(* CODESYS project SPT_EtherCat.library
   Author: SPT
   Version: 4.0.1
   Title: SPT EtherCat
   Placeholder: SPT EtherCat
   Company: Beckhoff Automation LLC

Project tree, tasks and I/O mapping:
  libraries: SPT Base Types, * (Beckhoff Automation LLC); SPT Event Logger, * (Beckhoff Automation LLC); Tc2_EtherCAT, * (Beckhoff Automation GmbH); Tc2_Standard, * (Beckhoff Automation GmbH); Tc2_System, * (Beckhoff Automation GmbH); Tc3_EventLogger, * (Beckhoff Automation GmbH); Tc3_Module, * (Beckhoff Automation GmbH)
  DUT/
    data type ST_EtherCatMaster_Command
    data type ST_EtherCatMaster_Config
    data type ST_EtherCatMaster_HMI
    data type ST_EtherCatMaster_Status
    data type ST_EtherCatMasterInfo
    data type ST_EtherCatSyncUnitTaskInfo
  Interface/
    interface I_EtherCatMaster: AmsNetIdEcMaster, ConfiguredSlaveCount, ConfiguredSlaveInfo, RegisterSyncUnit
    interface I_SyncUnitTask: IsHotConnect, NumberOfSlaves, SyncUnitName
  Project Information/
    function F_GetCompany [ST]
    function F_GetTitle [ST]
    function F_GetVersion [ST]
  Version/
    global variables Global_Version
  function block FB_Component_EtherCatMaster [ST]: CreateEvents, Monitoring, Reset, CyclicLogic, AmsNetIdEcMaster, ConfiguredSlaveCount, ConfiguredSlaveInfo, RegisterSyncUnit, FramesWcStatesOk, HMICommunication, Initialize, LookupMasterDevState, LookupSlaveDevState, MasterState, SlaveState
  function block FB_SyncUnitTask [ST]: CyclicLogic, IsHotConnect, NumberOfSlaves, SyncUnitName, FB_exit, FB_init, Initialize
  00000000-0000-0000-0000-000000000000|LICENSE
  LICENSE
  global variables Parameter_EtherCatMaster
*)

// DUT/ST_EtherCatMaster_Command
TYPE ST_EtherCatMaster_Command :
	STRUCT
	END_STRUCT
END_TYPE

// DUT/ST_EtherCatMaster_Config
TYPE ST_EtherCatMaster_Config :
	STRUCT
	END_STRUCT
END_TYPE

// DUT/ST_EtherCatMaster_HMI
TYPE ST_EtherCatMaster_HMI :
	STRUCT
		Config	: ST_EtherCatMaster_Config;
		Command : ST_EtherCatMaster_Command;
		Status	: ST_EtherCatMaster_Status;
	END_STRUCT
END_TYPE

// DUT/ST_EtherCatMaster_Status
TYPE ST_EtherCatMaster_Status :
	STRUCT
		AmsNetID			: T_AMSNETID;
		CfgSlaveCount		: UINT;
		EcSlavesState		: ARRAY[0..EC_MAX_SLAVES] OF ST_EcSlaveState;
		ConfiguredSlaveInfo : ARRAY[0..EC_MAX_SLAVES] OF ST_EcSlaveConfigData;
		EcSlaveTopologyInfo : ARRAY[0..EC_MAX_SLAVES] OF ST_TopologyDataEx;
	END_STRUCT
END_TYPE

// DUT/ST_EtherCatMasterInfo
TYPE ST_EtherCatMasterInfo :
	STRUCT
		AmsNetID	  AT %I* : AMSNETID;
		DevID		  AT %I* : UINT;
		DevState	  AT %I* : UINT;
		ChangeCount	  AT %I* : UINT;
		SlaveCount	  AT %I* : UINT;
		CfgSlaveCount AT %I* : UINT;
	END_STRUCT
END_TYPE

// DUT/ST_EtherCatSyncUnitTaskInfo
TYPE ST_EtherCatSyncUnitTaskInfo :
	STRUCT
		WcState	   AT %I* : BIT;
		ObjectId   AT %I* : OTCID;
		State	   AT %I* : UINT;
		SlaveCount AT %I* : UINT;
	END_STRUCT
END_TYPE

// Version/Global_Version
{attribute 'TcGenerated'}
{attribute 'no-analysis'}
{attribute 'linkalways'}
// This function has been automatically generated from the project information.
VAR_GLOBAL CONSTANT
	{attribute 'const_non_replaced'}
	stLibVersion_SPT_EtherCat : ST_LibVersion := (iMajor := 4, iMinor := 0, iBuild := 1, iRevision := 0, nFlags := 0, sVersion := '4.0.1');
END_VAR

// Parameter_EtherCatMaster
{attribute 'qualified_only'}
VAR_GLOBAL CONSTANT
	SYNC_UNIT_TASKS_PER_MASTER : UDINT := 10;	// Max Count of Sync Units per Master
	FRAMES_MAX				   : UDINT := 10;	// Max Count of Frames to Diagnose
	START_UP_TIME			   : TIME  := T#1S; // Time to Startup EtherCat Master Diagnostic at initial startup
END_VAR

// Interface/I_EtherCatMaster
INTERFACE I_EtherCatMaster EXTENDS I_ComponentBase

PROPERTY AmsNetIdEcMaster : T_AMSNETID
GET
END_GET
END_PROPERTY

PROPERTY ConfiguredSlaveCount : UINT
GET
END_GET
END_PROPERTY

PROPERTY ConfiguredSlaveInfo : REFERENCE TO ARRAY[0..EC_MAX_SLAVES] OF ST_EcSlaveConfigData
GET
END_GET
END_PROPERTY

METHOD RegisterSyncUnit : BOOL
VAR_INPUT
	ipSyncUnitTask : I_SyncUnitTask;
END_VAR
END_METHOD

END_INTERFACE

// Interface/I_SyncUnitTask
INTERFACE I_SyncUnitTask EXTENDS I_CyclicFB

PROPERTY IsHotConnect : BOOL
GET
END_GET
SET
END_SET
END_PROPERTY

PROPERTY PUBLIC NumberOfSlaves : UINT
GET
END_GET
END_PROPERTY

PROPERTY SyncUnitName : STRING(63)
GET
END_GET
END_PROPERTY

END_INTERFACE

// Project Information/F_GetCompany
// This function has been automatically generated from the project information.
{attribute 'signature_flag' := '1073741824'}
{attribute 'TcGenerated'}
{attribute 'no-analysis'}
FUNCTION F_GetCompany : WSTRING
VAR_INPUT
	
END_VAR

F_GetCompany := "Beckhoff Automation LLC";

END_FUNCTION

// Project Information/F_GetTitle
// This function has been automatically generated from the project information.
{attribute 'signature_flag' := '1073741824'}
{attribute 'TcGenerated'}
{attribute 'no-analysis'}
FUNCTION F_GetTitle : WSTRING
VAR_INPUT
	
END_VAR

F_GetTitle := "SPT EtherCat";

END_FUNCTION

// Project Information/F_GetVersion
// This function has been automatically generated from the project information.
{attribute 'signature_flag' := '1073741824'}
{attribute 'TcGenerated'}
{attribute 'no-analysis'}
FUNCTION F_GetVersion : ST_LibVersion
VAR_INPUT
	
END_VAR

F_GetVersion.iMajor := 4;
F_GetVersion.iMinor := 0;
F_GetVersion.iBuild := 1;
F_GetVersion.iRevision := 0;
F_GetVersion.sVersion := '4.0.1';
F_GetVersion.nFlags := 0;

END_FUNCTION

// FB_Component_EtherCatMaster
{attribute 'no_explicit_call' := 'do not call this POU directly'}
FUNCTION_BLOCK FB_Component_EtherCatMaster EXTENDS FB_ComponentBase IMPLEMENTS I_EtherCatMaster
VAR
	// Connections
	EtherCatMaster	   : ST_EtherCatMasterInfo;
	FrmXWcState AT %I* : ARRAY[0..(Parameter_EtherCatMaster.FRAMES_MAX - 1)] OF WORD; // link to task related ethercat frame state (Frm2WcState)

	// Internal Variables	
	_AmsNetIdEcMaster	 : T_AMSNETID;
	GetSlaveTopologyInfo : FB_EcGetSlaveTopologyInfo;
	EcGetAllSlaveStates	 : FB_EcGetAllSlaveStates;
	GetMasterFrameCount	 : FB_EcMasterFrameCount;
	LastFramesWcStatesOk : BOOL;
	EcSlavesState		 : ARRAY[0..EC_MAX_SLAVES] OF ST_EcSlaveState;
	EcSlaveTopologyInfo	 : ARRAY[0..EC_MAX_SLAVES] OF ST_TopologyDataEx;
	GetConfiguredSlaves	 : FB_EcGetConfSlaves;
	_ConfiguredSlaveInfo : ARRAY[0..EC_MAX_SLAVES] OF ST_EcSlaveConfigData;
	i					 : UDINT;

	// HMI
	EtherCatMaster_HMI : ST_EtherCatMaster_HMI;

	// Sync Units per Master
	SyncUnitTask : ARRAY[1..Parameter_EtherCatMaster.SYNC_UNIT_TASKS_PER_MASTER] OF I_SyncUnitTask;

	(*Sequence*)
	SlaveSeq			 : UINT;
	RunSlaveDiag		 : BOOL;
	LastChangeCount		 : UINT := 0;
	LastSlaveCount		 : UINT := 0;
	LastMasterState		 : UINT := 0;
	ErrorMaster			 : BOOL;
	WarningSlaveDisabled : BOOL;
	ErrorSlave			 : BOOL;
	FaultedSlave		 : UINT;

	// Alarms
	ComponentEtherCatDiagAlarms : ARRAY[1..COMPONENT_ETHERCAT_DIAG_ALARM_COUNT] OF FB_TcAlarm;
END_VAR

VAR CONSTANT
	COMPONENT_ETHERCAT_DIAG_ALARM_COUNT : UDINT := 20;
END_VAR

METHOD PROTECTED CreateEvents

// This method is called by Initialize() as required
F_CreateAllEventsInClass(Alarms		:= ComponentEtherCatDiagAlarms,
						 ClassSize	:= SIZEOF(TC_EVENTS.EtherCatDiagnostics),
						 pInitEvent := ADR(TC_EVENTS.EtherCatDiagnostics.InitReferenceEvent),
						 Prefix		:= Name);

SUPER^.CreateEvents();
END_METHOD

// Provides basic error detection and event handling for this component
METHOD PROTECTED Monitoring

// This method is called cyclically by CyclicLogic()
SUPER^.Monitoring();

(*EtherCat Messages*)
IF ErrorSlave AND (_ErrorId = 999) AND NOT ComponentEtherCatDiagAlarms[E_EtherCatDiagnostics.ReadSlave].bRaised THEN
	RaiseEventWithStrings(ComponentEtherCatDiagAlarms[E_EtherCatDiagnostics.ReadSlave], '', '');
ELSIF NOT ErrorSlave AND ComponentEtherCatDiagAlarms[E_EtherCatDiagnostics.ReadSlave].bRaised THEN
	ComponentEtherCatDiagAlarms[E_EtherCatDiagnostics.ReadSlave].Clear(0, 0);
END_IF

IF ErrorMaster AND NOT ComponentEtherCatDiagAlarms[E_EtherCatDiagnostics.MasterError].bRaised THEN
	RaiseAlarmWithStrings(ComponentEtherCatDiagAlarms[E_EtherCatDiagnostics.MasterError], LookupMasterDevState(EtherCatMaster.DevState), '');
END_IF

IF ErrorSlave AND NOT ComponentEtherCatDiagAlarms[E_EtherCatDiagnostics.SlaveError].bRaised THEN
	RaiseAlarmWithStrings(ComponentEtherCatDiagAlarms[E_EtherCatDiagnostics.SlaveError], _ConfiguredSlaveInfo[FaultedSlave].sName, LookupSlaveDevState(FaultedSlave));
END_IF

IF WarningSlaveDisabled AND NOT ComponentEtherCatDiagAlarms[E_EtherCatDiagnostics.SlaveDisabled].bRaised THEN
	RaiseEventWithStrings(ComponentEtherCatDiagAlarms[E_EtherCatDiagnostics.SlaveDisabled], '', '');
ELSIF NOT WarningSlaveDisabled AND ComponentEtherCatDiagAlarms[E_EtherCatDiagnostics.SlaveDisabled].bRaised THEN
	ComponentEtherCatDiagAlarms[E_EtherCatDiagnostics.SlaveDisabled].Clear(0, 0);
END_IF

_CurrentAlarmSeverity := F_GetMaxSeverityRaised(Alarms := ComponentEtherCatDiagAlarms, CurrentSeverity := _CurrentAlarmSeverity);
END_METHOD

// Clears error flags and error IDs for this component
METHOD PUBLIC Reset : BOOL
F_ClearAllEventsInClass(ComponentEtherCatDiagAlarms);
Reset				 := SUPER^.Reset();
WarningSlaveDisabled := FALSE;
LastMasterState		 := 0;
LastChangeCount		 := 0;
LastSlaveCount		 := 0;
_Error				 := FALSE;
_ErrorId			 := 0;
SlaveSeq			 := 0;
RunSlaveDiag		 := FALSE;
END_METHOD

// This method serves as the entry point for all underlying FB logic
METHOD PUBLIC CyclicLogic

// This method should be called cyclically by descendant function blocks by invoking SUPER^.CyclicLogic().  Alternatively, the contents of this method could be reimplemented entirely in which case a call to this method would not be necessary.
IF NOT _InitComplete THEN
	_InitComplete := Initialize();
	RETURN;
END_IF

(* Main Component Signals *)
IF _Simulate THEN
	_Busy	 := FALSE;
	_Error	 := FALSE;
	_ErrorId := 0;
ELSE
	// Initiate Detection of Change
	IF NOT _Busy THEN
		IF (LastChangeCount <> EtherCatMaster.ChangeCount) THEN // Master Change count changed
			RunSlaveDiag := TRUE;
		ELSIF ((EtherCatMaster.CfgSlaveCount <> EtherCatMaster.SlaveCount) AND (LastSlaveCount <> EtherCatMaster.SlaveCount)) THEN // Slave Count changed
			RunSlaveDiag := TRUE;
		ELSIF FramesWcStatesOk() <> LastFramesWcStatesOk THEN // Frame WC state changed
			RunSlaveDiag := TRUE;
		END_IF

		IF RunSlaveDiag THEN // Update Change
			LastChangeCount		 := EtherCatMaster.ChangeCount;
			LastSlaveCount		 := EtherCatMaster.SlaveCount;
			LastFramesWcStatesOk := FramesWcStatesOk();
		END_IF
	END_IF

	// Get slave topology info
	GetSlaveTopologyInfo(sNetId	  := _AmsNetIdEcMaster,
						 pAddrBuf := ADR(EcSlaveTopologyInfo),
						 cbBufLen := SIZEOF(EcSlaveTopologyInfo),
						 tTimeout := T#5S);

	// Get all slave states
	EcGetAllSlaveStates(sNetId	  := _AmsNetIdEcMaster,
						pStateBuf := ADR(EcSlavesState),
						cbBufLen  := SIZEOF(EcSlavesState),
						tTimeout  := T#5S);

	// Master State
	MasterState();

	// Slave State
	SlaveState();

	// SyncUnits
	FOR i := 1 TO Parameter_EtherCatMaster.SYNC_UNIT_TASKS_PER_MASTER DO
		IF SyncUnitTask[i] <> 0 THEN
			SyncUnitTask[i].CyclicLogic();
		END_IF
	END_FOR

	// Super
	_Busy  := SlaveSeq <> 0; // Sequence running
	_Error := _Error OR ErrorMaster OR ErrorSlave;
	SUPER^.CyclicLogic();
END_IF
END_METHOD

PROPERTY AmsNetIdEcMaster : T_AMSNETID
GET
AmsNetIdEcMaster := _AmsNetIdEcMaster;
END_GET
END_PROPERTY

PROPERTY ConfiguredSlaveCount : UINT
GET
ConfiguredSlaveCount := EtherCatMaster.CfgSlaveCount;
END_GET
END_PROPERTY

PROPERTY ConfiguredSlaveInfo : REFERENCE TO ARRAY[0..EC_MAX_SLAVES] OF ST_EcSlaveConfigData
GET
ConfiguredSlaveInfo REF= _ConfiguredSlaveInfo;
END_GET
END_PROPERTY

METHOD RegisterSyncUnit : BOOL
VAR_INPUT
	ipSyncUnitTask : I_SyncUnitTask;
END_VAR
FOR i := 1 TO Parameter_EtherCatMaster.SYNC_UNIT_TASKS_PER_MASTER DO
	IF SyncUnitTask[i] = 0 AND ipSyncUnitTask <> 0 THEN
		SyncUnitTask[i]	 := ipSyncUnitTask;
		RegisterSyncUnit := TRUE;
		RETURN;
	END_IF
END_FOR
END_METHOD

METHOD PROTECTED FramesWcStatesOk : BOOL
VAR_INPUT
END_VAR
FramesWcStatesOk := TRUE;
FOR i := 0 TO (GetMasterFrameCount.nFrames - 1) DO
	IF FrmXWcState[i] <> 0 THEN
		FramesWcStatesOk := FALSE;
		EXIT;
	END_IF
END_FOR
END_METHOD

// Provides interlocks for HMI control and updates HMI status information for this component
METHOD PROTECTED HMICommunication

// This method is called cyclically by CyclicLogic()
SUPER^.HMICommunication();

// Status
EtherCatMaster_HMI.Status.CfgSlaveCount		  := EtherCatMaster.CfgSlaveCount;
EtherCatMaster_HMI.Status.AmsNetID			  := _AmsNetIdEcMaster;
EtherCatMaster_HMI.Status.EcSlavesState		  := EcSlavesState;
EtherCatMaster_HMI.Status.ConfiguredSlaveInfo := ConfiguredSlaveInfo;
EtherCatMaster_HMI.Status.EcSlaveTopologyInfo := EcSlaveTopologyInfo;
END_METHOD

// Basic component initialization logic
METHOD PROTECTED Initialize : BOOL;
VAR_INST
	InitializeSequence : UINT := 0;
	Size			   : UDINT;
	StartupTime		   : TON;
END_VAR

// This method is called by CyclicLogic() as required
IF NOT _Error AND NOT (F_GetMappingStatus(ADR(EtherCatMaster.AmsNetID), SIZEOF(EtherCatMaster.AmsNetID)) <> EplcMappingStatus.MS_Unmapped) AND NOT _Simulate THEN
	_Error := TRUE;
	TRACE('Init Failed - AmsNetID mapped to Master!');
END_IF

IF NOT _Error AND NOT (F_GetMappingStatus(ADR(EtherCatMaster.DevID), SIZEOF(EtherCatMaster.DevID)) <> EplcMappingStatus.MS_Unmapped) AND NOT _Simulate THEN
	_Error := TRUE;
	TRACE('Init Failed - DevID mapped to Master!');
END_IF

IF NOT _Error AND NOT (F_GetMappingStatus(ADR(EtherCatMaster.DevState), SIZEOF(EtherCatMaster.DevState)) <> EplcMappingStatus.MS_Unmapped) AND NOT _Simulate THEN
	_Error := TRUE;
	TRACE('Init Failed - DevState mapped to Master!');
END_IF

IF NOT _Error AND NOT (F_GetMappingStatus(ADR(EtherCatMaster.ChangeCount), SIZEOF(EtherCatMaster.ChangeCount)) <> EplcMappingStatus.MS_Unmapped) AND NOT _Simulate THEN
	_Error := TRUE;
	TRACE('Init Failed - ChangeCount mapped to Master!');
END_IF

IF NOT _Error AND NOT (F_GetMappingStatus(ADR(EtherCatMaster.SlaveCount), SIZEOF(EtherCatMaster.SlaveCount)) <> EplcMappingStatus.MS_Unmapped) AND NOT _Simulate THEN
	_Error := TRUE;
	TRACE('Init Failed - CfgSlaveCount mapped to Master!');
END_IF

IF NOT _Error AND NOT (F_GetMappingStatus(ADR(EtherCatMaster.CfgSlaveCount), SIZEOF(EtherCatMaster.CfgSlaveCount)) <> EplcMappingStatus.MS_Unmapped) AND NOT _Simulate THEN
	_Error := TRUE;
	TRACE('Init Failed - CfgSlaveCount mapped to Master!');
END_IF

IF _Error THEN
	RETURN;
END_IF

IF _Simulate THEN
	Initialize := SUPER^.Initialize();
	RETURN;
END_IF

// Get all Slaves
_AmsNetIdEcMaster := F_CreateAmsNetId(EtherCatMaster.AmsNetID);
GetConfiguredSlaves(sNetId				:= _AmsNetIdEcMaster,
					pArrEcConfSlaveInfo := ADR(_ConfiguredSlaveInfo),
					cbBufLen			:= SIZEOF(_ConfiguredSlaveInfo),
					tTimeout			:= T#1S);

// Get Master Frames
GetMasterFrameCount(sNetId := _AmsNetIdEcMaster, tTimeout := T#1S);

// Init Sequence
CASE InitializeSequence OF
	(* Read Slave Info Data *)
	0:
		GetConfiguredSlaves.bExecute := TRUE;
		IF GetConfiguredSlaves.bBusy THEN
			InitializeSequence := InitializeSequence + 10;
		END_IF

	10:
		IF NOT GetConfiguredSlaves.bBusy AND NOT GetConfiguredSlaves.bError THEN
			InitializeSequence := InitializeSequence + 10;
		END_IF

		IF GetConfiguredSlaves.bError THEN
			_Error := TRUE;
			TRACE('Init Failed - Configured EtherCat Slaves could not be read - check linking of EtherCat Master FB!');
			InitializeSequence := 999;
		END_IF

	20: // Get Master Frame Count
		GetMasterFrameCount.bExecute := TRUE;
		IF GetMasterFrameCount.bBusy THEN
			InitializeSequence := InitializeSequence + 10;
		END_IF

	30:
		IF NOT GetMasterFrameCount.bBusy AND NOT GetMasterFrameCount.bError THEN
			// Check Frame Count
			IF GetMasterFrameCount.nFrames > Parameter_EtherCatMaster.FRAMES_MAX THEN
				_Error := TRUE;
				TRACE('Increase of Frame diagnostic array (Parameter_EtherCatMaster.FRAMES_MAX) and link to FrmXWcState!');
				RETURN;
			END_IF

			// Check Frame Linking
			FOR i := 0 TO (GetMasterFrameCount.nFrames - 1) DO
				IF NOT (F_GetMappingStatus(ADR(FrmXWcState[i]), SIZEOF(FrmXWcState[i])) <> EplcMappingStatus.MS_Unmapped) THEN
					_Error := TRUE;
					TRACE('Init Failed - FrmXWcState[x] not mapped to Master!');
					RETURN;
				END_IF
			END_FOR

			// 
			InitializeSequence := InitializeSequence + 10;
		END_IF

		IF GetMasterFrameCount.bError THEN
			_Error := TRUE;
			TRACE('Init Failed - Configured EtherCat Frames could not be read!');
			InitializeSequence := 999;
		END_IF

	40: // Startup time for Ethercat Master	
		StartupTime(IN := TRUE, PT := Parameter_EtherCatMaster.START_UP_TIME);
		IF StartupTime.Q THEN
			InitializeSequence := InitializeSequence + 10;
		END_IF

	50:
		Initialize := SUPER^.Initialize();
END_CASE
END_METHOD

METHOD PROTECTED LookupMasterDevState : STRING
VAR_INPUT
	State : UINT;
END_VAR
IF State.0 THEN
	LookupMasterDevState := 'Link error';
ELSIF State.1 THEN
	LookupMasterDevState := 'I/O locked after link error (I/O reset required)';
ELSIF State.2 THEN
	LookupMasterDevState := 'Link error (redundancy adapter)';
ELSIF State.3 THEN
	LookupMasterDevState := 'Missing one frame (redundancy mode)';
ELSIF State.4 THEN
	LookupMasterDevState := 'Out of send resources (I/O reset required)';
ELSIF State.5 THEN
	LookupMasterDevState := 'Watchdog triggered';
ELSIF State.6 THEN
	LookupMasterDevState := 'Ethernet driver (miniport) NOT found';
ELSIF State.7 THEN
	LookupMasterDevState := 'I/O reset active';
ELSIF State.8 THEN
	LookupMasterDevState := 'At least one device in INIT state';
ELSIF State.9 THEN
	LookupMasterDevState := 'At least one device in PRE-OP state';
ELSIF State.10 THEN
	LookupMasterDevState := 'At least one device in SAFE-OP state';
ELSIF State.11 THEN
	LookupMasterDevState := 'At least one device indicates an error state';
ELSIF State.12 THEN
	LookupMasterDevState := 'DC not in sync';
ELSE
	LookupMasterDevState := 'State not found';
END_IF
END_METHOD

METHOD PROTECTED LookupSlaveDevState : STRING
VAR_INPUT
	Slave : UINT;
END_VAR

VAR_INST
	DiagByte	: BYTE;
	BitMaskDiag : BYTE := 16#0F;
END_VAR
//_____________________________________________________________________________________________________

(* State *)
BitMaskDiag := 16#0F;
DiagByte	:= EcSlavesState[Slave].deviceState AND BitMaskDiag;
CASE DiagByte OF
	EC_DEVICE_STATE_INIT:
		LookupSlaveDevState := 'Init';

	EC_DEVICE_STATE_PREOP:
		LookupSlaveDevState := 'Pre-op';

	EC_DEVICE_STATE_BOOTSTRAP:
		LookupSlaveDevState := 'Boot';

	EC_DEVICE_STATE_SAFEOP:
		LookupSlaveDevState := 'Safe-op';

	EC_DEVICE_STATE_OP:
		LookupSlaveDevState := 'OP';

ELSE
	LookupSlaveDevState := '';
END_CASE

(* Additional State Bits *)
IF EcSlavesState[Slave].deviceState.4 THEN // EC_DEVICE_STATE_ERROR
	LookupSlaveDevState := CONCAT(LookupSlaveDevState, ' - ');
	LookupSlaveDevState := CONCAT(LookupSlaveDevState, 'State machine error in the EtherCAT slave');
END_IF

IF EcSlavesState[Slave].deviceState.5 THEN // EC_DEVICE_STATE_INVALID_VPRS
	LookupSlaveDevState := CONCAT(LookupSlaveDevState, ' - ');
	LookupSlaveDevState := CONCAT(LookupSlaveDevState, 'Invalid vendor ID');
END_IF

IF EcSlavesState[Slave].deviceState.6 THEN // EC_DEVICE_STATE_INITCMD_ERROR
	LookupSlaveDevState := CONCAT(LookupSlaveDevState, ' - ');
	LookupSlaveDevState := CONCAT(LookupSlaveDevState, 'Error during sending of initialization commands');
END_IF

IF EcSlavesState[Slave].deviceState.7 THEN // EC_DEVICE_STATE_DISABLED
	LookupSlaveDevState := CONCAT(LookupSlaveDevState, ' - ');
	LookupSlaveDevState := CONCAT(LookupSlaveDevState, 'Slave is disabled');
END_IF

//_____________________________________________________________________________________________________

(* Link States *)
IF EcSlavesState[Slave].linkState.0 THEN // EC_LINK_STATE_NOT_PRESENT
	LookupSlaveDevState := CONCAT(LookupSlaveDevState, ' - ');
	LookupSlaveDevState := CONCAT(LookupSlaveDevState, 'No EtherCAT communication with the EtherCAT slave');
END_IF

IF EcSlavesState[Slave].linkState.1 THEN // EC_LINK_STATE_LINK_WITHOUT_COMM
	LookupSlaveDevState := CONCAT(LookupSlaveDevState, ' - ');
	LookupSlaveDevState := CONCAT(LookupSlaveDevState, 'Error AT port X');
END_IF

IF EcSlavesState[Slave].linkState.2 THEN // EC_LINK_STATE_MISSING_LINK
	LookupSlaveDevState := CONCAT(LookupSlaveDevState, ' - ');
	LookupSlaveDevState := CONCAT(LookupSlaveDevState, 'Missing link AT port X');
END_IF

IF EcSlavesState[Slave].linkState.3 THEN // EC_LINK_STATE_ADDITIONAL_LINK
	LookupSlaveDevState := CONCAT(LookupSlaveDevState, ' - ');
	LookupSlaveDevState := CONCAT(LookupSlaveDevState, 'Additional link AT port X');
END_IF

(* Additional State Bits *)
IF EcSlavesState[Slave].linkState.4 THEN // EC_LINK_STATE_PORT_A
	LookupSlaveDevState := CONCAT(LookupSlaveDevState, ' - ');
	LookupSlaveDevState := CONCAT(LookupSlaveDevState, 'Port 0');
END_IF

IF EcSlavesState[Slave].linkState.5 THEN // EC_LINK_STATE_PORT_B
	LookupSlaveDevState := CONCAT(LookupSlaveDevState, ' - ');
	LookupSlaveDevState := CONCAT(LookupSlaveDevState, 'Port 1');
END_IF

IF EcSlavesState[Slave].linkState.6 THEN // EC_LINK_STATE_PORT_C
	LookupSlaveDevState := CONCAT(LookupSlaveDevState, ' - ');
	LookupSlaveDevState := CONCAT(LookupSlaveDevState, 'Port 2');
END_IF

IF EcSlavesState[Slave].linkState.7 THEN // EC_LINK_STATE_PORT_D
	LookupSlaveDevState := CONCAT(LookupSlaveDevState, ' - ');
	LookupSlaveDevState := CONCAT(LookupSlaveDevState, 'Port 3');
END_IF
END_METHOD

METHOD PROTECTED MasterState : BOOL
VAR_INPUT
END_VAR
IF (LastMasterState <> EtherCatMaster.DevState) AND (EtherCatMaster.DevState <> 0) AND (EtherCatMaster.SlaveCount < EtherCatMaster.CfgSlaveCount) THEN
	IF EtherCatMaster.DevState <> 0 THEN // Error in Master
		ErrorMaster := TRUE;
		_ErrorId	:= EtherCatMaster.DevState;
	END_IF
ELSE
	ErrorMaster := FALSE;
END_IF
END_METHOD

METHOD PROTECTED SlaveState : BOOL
VAR_INST
	DiagByte	: BYTE;
	BitMaskDiag : BYTE := 16#0F;
END_VAR
CASE SlaveSeq OF
	(* Wait for start *)
	0:
		EcGetAllSlaveStates.bExecute  := FALSE;
		GetConfiguredSlaves.bExecute  := FALSE;
		GetSlaveTopologyInfo.bExecute := FALSE;
		IF RunSlaveDiag THEN
			RunSlaveDiag		 := FALSE;
			ErrorSlave			 := FALSE; // Reset for re-check
			WarningSlaveDisabled := FALSE;
			SlaveSeq			 := SlaveSeq + 10;
		END_IF

	(* Update Topology*)
	10:
		GetSlaveTopologyInfo.bExecute := TRUE;
		IF GetSlaveTopologyInfo.bBusy THEN
			SlaveSeq := SlaveSeq + 10;
		END_IF

	20:
		IF NOT GetSlaveTopologyInfo.bBusy AND NOT GetSlaveTopologyInfo.bError THEN
			SlaveSeq := SlaveSeq + 10;
		END_IF

		IF GetSlaveTopologyInfo.bError THEN
			SlaveSeq := 999;
		END_IF

	(* Read Slave States *)
	30:
		EcGetAllSlaveStates.bExecute := TRUE;
		IF EcGetAllSlaveStates.bBusy THEN
			SlaveSeq := SlaveSeq + 10;
		END_IF

	40:
		IF NOT EcGetAllSlaveStates.bBusy AND NOT EcGetAllSlaveStates.bError THEN
			SlaveSeq := SlaveSeq + 10;
		END_IF

		IF EcGetAllSlaveStates.bError THEN
			SlaveSeq := 999;
		END_IF

	(* Evaluate Slave Error *)
	50:
		FOR FaultedSlave := 0 TO (EtherCatMaster.CfgSlaveCount - 1) DO
			BitMaskDiag := 16#0F;
			DiagByte	:= EcSlavesState[FaultedSlave].deviceState AND BitMaskDiag;
			IF DiagByte <> EC_DEVICE_STATE_OP AND EcSlaveTopologyInfo[FaultedSlave].nStatusBits.4 = FALSE THEN // No error if hotconnect
				IF EcSlavesState[FaultedSlave].deviceState.7 THEN											   // Slave is Disabled - warning only
					WarningSlaveDisabled := TRUE;
				ELSE
					ErrorSlave := TRUE;
					EXIT;
				END_IF
			END_IF

			BitMaskDiag := 16#0F;
			DiagByte	:= EcSlavesState[FaultedSlave].linkState AND BitMaskDiag;
			IF DiagByte <> EC_LINK_STATE_OK AND EcSlaveTopologyInfo[FaultedSlave].nStatusBits.4 = FALSE THEN // Next slave is in hotconnect group, no error
				ErrorSlave := TRUE;
				EXIT;
			END_IF
		END_FOR

		SlaveSeq := SlaveSeq + 10;

	60:
		SlaveSeq := 0;

	(* Sequence Error*)
	999:
		ErrorSlave := TRUE;
		_ErrorId   := 999;
		SlaveSeq   := 0;
END_CASE
END_METHOD

END_FUNCTION_BLOCK

// FB_SyncUnitTask
{attribute 'no_explicit_call' := 'do not call this POU directly'}
FUNCTION_BLOCK FINAL FB_SyncUnitTask EXTENDS FB_CyclicFB IMPLEMENTS I_SyncUnitTask
VAR
	// IO to Sync Unit Task configuration
	SyncUnitTaskInfo : ST_EtherCatSyncUnitTaskInfo;

	// Internal Variables
	EcGetAllSyncUnitSlaveAddr : FB_EcGetAllSyncUnitSlaveAddr;
	SyncUnitSlaveAddresses	  : POINTER TO UINT;
	SyncUnitSlaveNames		  : POINTER TO STRING(31);
	SyncUnitState			  : (SYNC_UNIT_OK,
		READ_SLAVES,
		POPULATE_SLAVE_NAMES,
		WORKING_COUNTER_ERROR,
		READ_ERROR) := SYNC_UNIT_OK;
	i : UDINT; // Iterator
	j : UDINT; // Iterator

	// Properties
	_SyncUnitName	: STRING(63);
	_NumberOfSlaves : UINT;
	_IsHotConnect	: BOOL;

	// Connection to EtherCat Master
	ipEtherCatMaster : I_EtherCatMaster;

	// Alarm
	SyncUnitAlarm : ARRAY[1..SYNC_UNIT_ALARM_MAX] OF FB_TcAlarm;
END_VAR

VAR
	// Build slave in sync unit collection to display, string limit to 80
	TempSlaveMessage  : STRING;
	SlaveMessagePartA : STRING;
	SlaveMessagePartB : STRING;
END_VAR

VAR CONSTANT
	ERROR_READ_SLAVE_NAMES	   : UDINT := 1;
	ERROR_REGISTER_SYNC_UNIT   : UDINT := 2;
	ERROR_VALID_DATA_SYNC_UNIT : UDINT := 3;
	STRING_LEN				   : INT   := 80;
	SYNC_UNIT_ALARM_MAX		   : UINT  := 3;
END_VAR

METHOD PUBLIC CyclicLogic
VAR_INPUT
END_VAR

VAR_INST
	tempSlaveInfo : REFERENCE TO ARRAY[0..EC_MAX_SLAVES] OF ST_EcSlaveConfigData;
END_VAR
IF NOT _InitComplete THEN
	_InitComplete := Initialize();
	RETURN;
END_IF

// Read SyncUnit Slave Names
tempSlaveInfo REF= ipEtherCatMaster.ConfiguredSlaveInfo;
EcGetAllSyncUnitSlaveAddr(sNetId	:= '',
						  nObjectId := SyncUnitTaskInfo.ObjectId,
						  pAddrBuf	:= SyncUnitSlaveAddresses,
						  cbBufLen	:= (SIZEOF(UINT) * SyncUnitTaskInfo.SlaveCount),
						  tTimeout	:= T#5S,
						  nSlaves	=> _NumberOfSlaves);

EcGetAllSyncUnitSlaveAddr.bExecute := FALSE;

// Sync Unit States
CASE SyncUnitState OF
	SYNC_UNIT_OK: // Working counter error detected on this sync unit
		IF SyncUnitTaskInfo.WcState THEN
			SyncUnitSlaveAddresses			   := __NEW(UINT, SyncUnitTaskInfo.SlaveCount);
			SyncUnitState					   := READ_SLAVES;
			EcGetAllSyncUnitSlaveAddr.bExecute := TRUE;
			SUPER^._Busy					   := TRUE;
		ELSE
			SUPER^._Error	:= FALSE;
			SUPER^._ErrorID := 0;
			SUPER^._Busy	:= FALSE;
		END_IF

	READ_SLAVES: // Read Slave address in Sync Unit
		IF NOT EcGetAllSyncUnitSlaveAddr.bBusy AND NOT EcGetAllSyncUnitSlaveAddr.bError AND (_NumberOfSlaves > 0) THEN
			SyncUnitState := POPULATE_SLAVE_NAMES;
		END_IF

		IF (EcGetAllSyncUnitSlaveAddr.bError OR (_NumberOfSlaves = 0)) AND NOT EcGetAllSyncUnitSlaveAddr.bBusy THEN
			SyncUnitState := READ_ERROR;
		END_IF

	POPULATE_SLAVE_NAMES: // Populate Names
		IF SyncUnitSlaveNames = 0 THEN
			SyncUnitSlaveNames := __NEW(STRING(31), _NumberOfSlaves);
		END_IF

		FOR i := 0 TO (_NumberOfSlaves - 1) DO
			FOR j := 0 TO (ipEtherCatMaster.ConfiguredSlaveCount - 1) DO
				IF SyncUnitSlaveAddresses[i] <> 0 THEN
					IF SyncUnitSlaveAddresses[i] = tempSlaveInfo[j].nAddr THEN
						SyncUnitSlaveNames[i] := tempSlaveInfo[j].sName;
					END_IF
				END_IF
			END_FOR
		END_FOR

		TempSlaveMessage  := '';
		SlaveMessagePartA := '';
		SlaveMessagePartB := '';
		FOR j := 0 TO (_NumberOfSlaves - 1) DO
			IF LEN(SyncUnitSlaveNames[j]) > 0 THEN
				TempSlaveMessage := CONCAT(SyncUnitSlaveNames[j], ', ');
				IF (LEN(TempSlaveMessage) + LEN(SlaveMessagePartA)) <= STRING_LEN THEN
					SlaveMessagePartA := CONCAT(SlaveMessagePartA, TempSlaveMessage);
				ELSIF (LEN(TempSlaveMessage) + LEN(SlaveMessagePartB)) <= STRING_LEN THEN
					SlaveMessagePartB := CONCAT(SlaveMessagePartB, TempSlaveMessage);
				END_IF
			END_IF
		END_FOR

		__DELETE(SyncUnitSlaveAddresses);
		__DELETE(SyncUnitSlaveNames);
		SyncUnitState := WORKING_COUNTER_ERROR;

	WORKING_COUNTER_ERROR: // Wait for Sync Unit valid data
		SUPER^._Busy	:= FALSE;
		SUPER^._Error	:= TRUE;
		SUPER^._ErrorID := ERROR_VALID_DATA_SYNC_UNIT;

		// Raise Error-Warning
		IF _IsHotConnect AND NOT SyncUnitAlarm[E_SyncUnit.SyncUnitWarning].bRaised THEN
			F_RaiseAlarmWithStringParameters(Alarm	  := SyncUnitAlarm[E_SyncUnit.SyncUnitWarning],
											 String_1 := CONCAT(ipEtherCatMaster.Name, CONCAT(' - ', _SyncUnitName)),
											 String_2 := SlaveMessagePartA,
											 String_3 := SlaveMessagePartB);
		ELSIF NOT _IsHotConnect AND NOT SyncUnitAlarm[E_SyncUnit.SyncUnitError].bRaised THEN
			F_RaiseAlarmWithStringParameters(Alarm	  := SyncUnitAlarm[E_SyncUnit.SyncUnitError],
											 String_1 := CONCAT(ipEtherCatMaster.Name, CONCAT(' - ', _SyncUnitName)),
											 String_2 := SlaveMessagePartA,
											 String_3 := SlaveMessagePartB);
		END_IF

		// Wait for WC OK
		IF NOT SyncUnitTaskInfo.WcState THEN
			F_ClearAllEventsInClass(SyncUnitAlarm);
			SyncUnitState := SYNC_UNIT_OK;
		END_IF

	READ_ERROR: // Error
		TRACE(CONCAT('Sync Unit Slave Names could not be read! Error ID: ', TO_STRING(EcGetAllSyncUnitSlaveAddr.nErrId)));
		SUPER^._Error	:= TRUE;
		SUPER^._ErrorID := ERROR_READ_SLAVE_NAMES;
		__DELETE(SyncUnitSlaveAddresses);
		__DELETE(SyncUnitSlaveNames);
		SyncUnitState := SYNC_UNIT_OK;
END_CASE
END_METHOD

PROPERTY IsHotConnect : BOOL
GET
IsHotConnect := _IsHotConnect;
END_GET
SET
_IsHotConnect := IsHotConnect;
END_SET
END_PROPERTY

PROPERTY PUBLIC NumberOfSlaves : UINT
GET
NumberOfSlaves := _NumberOfSlaves;
END_GET
END_PROPERTY

PROPERTY SyncUnitName : STRING(63)
GET
SyncUnitName := _SyncUnitName;
END_GET
END_PROPERTY

METHOD FB_exit : BOOL
VAR_INPUT
	bInCopyCode : BOOL; // if TRUE, the exit method is called for exiting an instance that is copied afterwards (online change).
END_VAR
__DELETE(SyncUnitSlaveAddresses);
__DELETE(SyncUnitSlaveNames);
END_METHOD

METHOD FB_init : BOOL
VAR_INPUT
	bInitRetains   : BOOL;			   // if TRUE, the retain variables are initialized (warm start / cold start)
	bInCopyCode	   : BOOL;			   // if TRUE, the instance afterwards gets moved into the copy code (online change)
	EtherCatMaster : I_EtherCatMaster; // Assign EtherCat Master for this Sync Unit
END_VAR
IF EtherCatMaster <> 0 THEN
	IF EtherCatMaster.RegisterSyncUnit(THIS^) THEN
		ipEtherCatMaster := EtherCatMaster;
	ELSE
		SUPER^._Error	:= TRUE;
		SUPER^._ErrorID := ERROR_REGISTER_SYNC_UNIT;
	END_IF
END_IF
END_METHOD

METHOD PRIVATE Initialize : BOOL
VAR_INPUT
END_VAR
// Check valid Pointers
IF ipEtherCatMaster = 0 THEN
	_Error	 := TRUE;
	_ErrorId := 999;
	TRACE('SyncUnit missing EtherCat Master reference!');
	RETURN;
END_IF

// Check Linking
IF NOT _Error AND NOT (F_GetMappingStatus(ADR(SyncUnitTaskInfo.ObjectId), SIZEOF(SyncUnitTaskInfo.ObjectId)) <> EplcMappingStatus.MS_Unmapped) THEN
	_Error := TRUE;
	TRACE('Init Failed - SyncUnitTaskInfo.ObjectId mapped to SyncUnit Diagnostic!');
END_IF

IF NOT _Error AND NOT (F_GetMappingStatus(ADR(SyncUnitTaskInfo.SlaveCount), SIZEOF(SyncUnitTaskInfo.SlaveCount)) <> EplcMappingStatus.MS_Unmapped) THEN
	_Error := TRUE;
	TRACE('Init Failed - SyncUnitTaskInfo.SlaveCount mapped to SyncUnit Diagnostic!');
END_IF

IF NOT _Error AND NOT (F_GetMappingStatus(ADR(SyncUnitTaskInfo.State), SIZEOF(SyncUnitTaskInfo.State)) <> EplcMappingStatus.MS_Unmapped) THEN
	_Error := TRUE;
	TRACE('Init Failed - SyncUnitTaskInfo.State mapped to SyncUnit Diagnostic!');
END_IF

IF NOT _Error AND NOT (F_GetMappingStatus(ADR(SyncUnitTaskInfo.WcState), SIZEOF(SyncUnitTaskInfo.WcState)) <> EplcMappingStatus.MS_Unmapped) THEN
	_Error := TRUE;
	TRACE('Init Failed - SyncUnitTaskInfo.WcState mapped to SyncUnit Diagnostic!');
END_IF

IF _Error THEN
	RETURN;
END_IF

// Get SyncUnit Name
F_EcGetSyncUnitName(SyncUnitTaskInfo.ObjectId, sSyncUnitName => _SyncUnitName);

// Create Events
F_CreateAllEventsInClass(Alarms		:= SyncUnitAlarm,
						 ClassSize	:= SIZEOF(TC_EVENTS.SyncUnit),
						 pInitEvent := ADR(TC_EVENTS.SyncUnit.InitReferenceEvent),
						 Prefix		:= _SyncUnitName);

Initialize := TRUE;
END_METHOD

END_FUNCTION_BLOCK
